Universal Robots PolyScope program: Bridge_flat_roof.urp

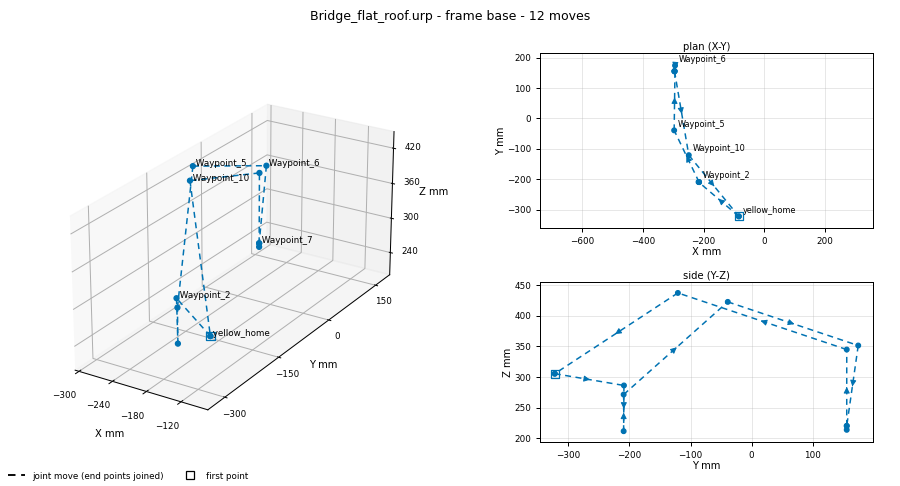
[picture p0: tool path of Bridge_flat_roof.urp in frame base, 12 of 12 moves have a stored position in this frame; points joined in program order, loops and branches not executed]
Program Bridge_flat_roof (installation=default directory=/programs/usbdisk/Zahra createdIn=5.11.11.1010533 lastSavedIn=5.11.11.1010533 robotSerialNumber=20205300864)
Calibrated DH parameters: a=[-0.000166, -0.243494, -0.153108, 0.000057, -0.000123, 0]; d=[0.151897, -1.34267, 53.988124, -52.514559, 0.085283, 0.092193]; alpha=[1.572472, -0.003756, 0.002824, 1.570807, -1.572621, 0]; deltaTheta=[0, 0.020704, 7.033215, -0.770746, 0.000004, 0]
Robot Program (runOnlyOnce=true)
  MoveJ speed 60 deg/s, acceleration 80 deg/s^2 (useActiveTCP=true) feature=Base
    Waypoint yellow_home: TCP in base x=-84.299 y=-321.875 z=305.481 mm, rx=-2.0809 ry=-2.2572 rz=0.0984 rad; joints [-79.978, -91.201, -87.971, -91.7, 84.671, 815.506] deg
    Waypoint Waypoint_2: TCP in base x=-216.822 y=-208.813 z=286.218 mm, rx=-2.2946 ry=-2.1457 rz=-0.0076 rad; joints [-110.448, -83.773, -100.41, -85.96, 90.176, 793.504] deg
    URCap Gripper (Robotiq_Grippers, Robotiq Inc.) dataModel(position=27.84313725490196, force=94.0, speed=40.0, positionInDouble=27.84313725490196, forceInDouble=94.0, speedInDouble=40.0, slaveIds=[9], blocking=true, robotCompliant=false)
    Waypoint Waypoint_3: TCP in base x=-215.062 y=-209.285 z=211.444 mm, rx=2.2181 ry=2.2017 rz=0.0234 rad; joints [-110.46, -88.495, -116.903, -64.884, 91.273, 790.128] deg
    URCap Gripper (Robotiq_Grippers, Robotiq Inc.) dataModel(position=58.549019607843135, force=94.0, speed=40.0, positionInDouble=58.549019607843135, forceInDouble=94.0, speedInDouble=40.0, slaveIds=[9], blocking=true, robotCompliant=false)
    Waypoint Waypoint_4: TCP in base x=-215.049 y=-209.29 z=271.375 mm, rx=2.218 ry=2.2017 rz=0.0235 rad; joints [-110.437, -84.156, -104.035, -82.093, 91.269, 790.103] deg
    Waypoint Waypoint_5: TCP in base x=-297.018 y=-39.057 z=422.848 mm, rx=-2.029 ry=-2.3286 rz=0.0527 rad; joints [-145.791, -89.676, -57.597, -119.966, 87.529, 746.337] deg
    Waypoint Waypoint_6: TCP in base x=-294.082 y=174.18 z=351.52 mm, rx=2.0996 ry=2.3336 rz=-0.0191 rad; joints [-188.369, -95.37, -71.421, -102.831, 90.631, 705.669] deg
    Waypoint Waypoint_7: TCP in base x=-295.834 y=155.405 z=220.145 mm, rx=2.2314 ry=2.1767 rz=0.0385 rad; joints [-184.724, -96.392, -105.334, -70.141, 89.876, 716.85] deg
    Waypoint Waypoint_8: TCP in base x=-295.834 y=155.39 z=213.704 mm, rx=2.2313 ry=2.1767 rz=0.0387 rad; joints [-184.723, -96.997, -106.511, -68.366, 89.875, 716.855] deg
    URCap Gripper (Robotiq_Grippers, Robotiq Inc.) dataModel(position=25.098039215686274, force=94.0, speed=40.0, positionInDouble=25.098039215686274, forceInDouble=94.0, speedInDouble=40.0, slaveIds=[9], blocking=true, robotCompliant=false)
    Waypoint Waypoint_7: TCP in base x=-295.834 y=155.405 z=220.145 mm, rx=2.2314 ry=2.1767 rz=0.0385 rad; joints [-184.724, -96.392, -105.334, -70.141, 89.876, 716.85] deg
    Waypoint Waypoint_9: TCP in base x=-295.826 y=155.403 z=344.932 mm, rx=2.2313 ry=2.1768 rz=0.0385 rad; joints [-184.667, -93.949, -73.888, -104.03, 89.825, 716.835] deg
    Waypoint Waypoint_10: TCP in base x=-248.907 y=-120.638 z=437.46 mm, rx=1.2966 ry=2.836 rz=-0.3231 rad; joints [-127.018, -82.018, -64.585, -111.808, 92.861, 732.466] deg
    Waypoint yellow_home: TCP in base x=-84.299 y=-321.875 z=305.481 mm, rx=-2.0809 ry=-2.2572 rz=0.0984 rad; joints [-79.978, -91.201, -87.971, -91.7, 84.671, 815.506] deg
